PROGRAM Main_Read
VAR
	TimeStr	: STRING;
END_VAR

(* get timestamp *)
TimeStr	:= Background_Time.TimeStr;

(* read sensors *)
Read_IMU();
//Read_FatigueCam();
Read_GPS();
Read_Payload();
Read_Pressure();
Read_Strain();

END_PROGRAM

(* stored: Version 1.1.0.1, ProductVersion 3.1.4024.6
   POU Main_Read: Id {a2a7af55-88d8-4c94-9be8-8a85ac14953c}, SpecialFunc None *)
